FUNCTION_BLOCK MoveAbsoluteTask EXTENDS TcoCore.TcoTask IMPLEMENTS ITcoDriveSimple
VAR
    {attribute addProperty Name "<#Position#>"}
    _position : LREAL;
    {attribute addProperty Name "<#Velocity#>"}
    _velocity : LREAL;
    {attribute addProperty Name "<#Acceleration#>"}
    _acceleration : LREAL;
    {attribute addProperty Name "<#Deceleration#>"}
    _deceleration : LREAL;
    {attribute addProperty Name "<#Jerk#>"}
    _jerk : LREAL;
END_VAR
VAR
    {attribute 'hide'}
    _axisRef : REFERENCE TO TcoAxisRef;
    {attribute 'hide'}
    _mcMoveAbsolute : Tc2_MC2.MC_MoveAbsolute;
    {attribute 'hide'}
    _mcMoveAbsolutePreconditionOK : BOOL;
    {attribute 'hide'}
	_mcReadAxisEncoderReferenceSystem : MC_ReadParameter;
	
	_AxisEncoderReferenceSystem : eAxisEncoderReferenceSystem;
END_VAR

IF NOT __ISVALIDREF(_axisRef) THEN
    IF __ISVALIDREF(DriveRef) THEN
        _axisRef REF= DriveRef.AxisRef;
    ELSE
        RETURN;
    END_IF
END_IF

IF Execute() THEN
    _mcReadAxisEncoderReferenceSystem(Axis := _axisRef,
        Enable := TRUE,
        ParameterNumber := eAxisParameter.AxisEncoderReferenceSystem,
        ReadMode := Tc2_MC2.E_ReadMode.READMODE_ONCE);

    IF _mcReadAxisEncoderReferenceSystem.Valid THEN
        LREAL_TO_Tco_AxisEncoderReferenceSystem(_mcReadAxisEncoderReferenceSystem.Value, _AxisEncoderReferenceSystem);

        IF _AxisEncoderReferenceSystem = eAxisEncoderReferenceSystem.ABSOLUTE OR
            _AxisEncoderReferenceSystem = eAxisEncoderReferenceSystem.ABSOLUTE_MODULO OR
            _AxisEncoderReferenceSystem = eAxisEncoderReferenceSystem.ABSOLUTE_MULTITURN OR
            _AxisEncoderReferenceSystem = eAxisEncoderReferenceSystem.ABSOLUTE_SINGLETURN THEN
            _mcMoveAbsolutePreconditionOK := TRUE;
        ELSE
            _mcMoveAbsolutePreconditionOK := _axisRef.Status.Homed;
        END_IF
    END_IF

    IF NOT DriveRef._movementState.MovePreconditionsOk(THIS^, _mcMoveAbsolutePreconditionOK) THEN
        IF _mcReadAxisEncoderReferenceSystem.Valid AND NOT _mcMoveAbsolutePreconditionOK THEN
            Messenger.Error('Move absolute not possible as axis is Incremental and not Homed');
        END_IF

        RETURN;
    END_IF

    _mcMoveAbsolute(Axis := _axisRef,
        Execute := NOT _mcMoveAbsolute.Busy,
        Position := _position,
        Velocity := _velocity,
        Acceleration := _acceleration,
        Deceleration := _deceleration,
        Jerk := _jerk,
        BufferMode := Tc2_MC2.MC_Aborting,
        Done =>,
        Busy =>,
        Active =>,
        CommandAborted =>,
        Error =>,
        ErrorID =>);

    IF _mcMoveAbsolute.CommandAborted THEN
        THIS^.Abort();
    END_IF

    DoneWhen(_mcMoveAbsolute.Done);
    ThrowWhen(_mcMoveAbsolute.Error);
END_IF

PROPERTY DriveRef : REFERENCE TO TcoDriveSimple
GET
VAR
    _drive : ITcoDriveSimple := 0;
END_VAR
IF __QUERYINTERFACE(THIS^.Parent, _drive) THEN
    DriveRef REF= _drive.DriveRef;
END_IF
END_GET
END_PROPERTY

METHOD PUBLIC FB_init : BOOL
VAR_INPUT
    bInitRetains : BOOL; // if TRUE, the retain variables are initialized (warm start / cold start)
    bInCopyCode : BOOL; // if TRUE, the instance afterwards gets moved into the copy code (online change)
  	ParentObject : ITcoObject;	
END_VAR
END_METHOD

METHOD INTERNAL InvokeWithParams : ITcoTaskStatus
VAR_INPUT
    inPosition : LREAL;
    inVelocity : LREAL;
    inAcceleration : LREAL;
    inDeceleration : LREAL;
    inJerk : LREAL;
END_VAR
_position := inPosition;
_velocity := inVelocity;
_acceleration := inAcceleration;
_deceleration := inDeceleration;
_jerk := inJerk;
InvokeWithParams := THIS^.Invoke();
END_METHOD

(*~
	<docu>
		<summary>
			Executes when task is aborted.
		</summary>			
	</docu>	
~*)
METHOD PROTECTED OnAbort
IF NOT __ISVALIDREF(_axisRef) THEN
    IF __ISVALIDREF(DriveRef) THEN
        _axisRef REF= DriveRef.AxisRef;
    ELSE
        RETURN;
    END_IF
END_IF

THIS^.DriveRef.Stop(-1, -1);
_mcMoveAbsolute(Axis := _axisRef, Execute := FALSE);
_mcReadAxisEncoderReferenceSystem(Axis :=_axisRef,Enable := FALSE);
THIS^.DriveRef._movementState.Restore();
END_METHOD

(*~
	<docu>
		<summary>
			Executes when task reaches the ```Done``` state .
		</summary>			
	</docu>	
~*)
METHOD PROTECTED OnDone
_mcMoveAbsolute(Axis := _axisRef, Execute := FALSE);
_mcReadAxisEncoderReferenceSystem(Axis :=_axisRef,Enable := FALSE);
THIS^.DriveRef._movementState.Restore();
END_METHOD

(*~
	<docu>
		<summary>
			Executes when task reaches the ```Error``` state.
			<para>
				Do not confuse with <see cref="PlcDocu.TcoCore.TcoTask.WhileError()"/>, that is called cyclically until '''Error''' state is left.
			</para>
		</summary>			
	</docu>	
~*)
METHOD PROTECTED OnError
THIS^.DriveRef._movementState.Restore();

IF NOT _axisRef.Status.Error THEN
	DriveRef.SetErrorID( DriveRef._moveAbsoluteTask._mcMoveAbsolute.ErrorID);
END_IF
_mcMoveAbsolute(Axis := _axisRef, Execute := FALSE);
_mcReadAxisEncoderReferenceSystem(Axis :=_axisRef,Enable := FALSE);
END_METHOD

METHOD PROTECTED OnStart
_mcMoveAbsolute(Axis := _axisRef, Execute := FALSE);
_mcReadAxisEncoderReferenceSystem(Axis :=_axisRef,Enable := FALSE);
END_METHOD

(*~
	<docu>
		<summary>
			Restores this instance to the Ready state. Can be called explicitly or from within one of the restore mechanisms.
			<para>
				See also <see cref="PlcDocu.TcoCore.TcoTask.AutoRestorable()"/>
			</para>
		</summary>			
	</docu>	
~*)
METHOD Restore : ITcoRestorable
SUPER^.Restore();
END_METHOD

(*~
	<docu>
		<summary>
			Executes until task is in ```Error``` state .
		</summary>			
	</docu>	
~*)
METHOD PROTECTED WhileError
IF NOT _axisRef.Status.Error THEN
	DriveRef.SetErrorID( DriveRef._moveAbsoluteTask._mcMoveAbsolute.ErrorID);
    _mcMoveAbsolute(Axis := _axisRef, Execute := FALSE);
END_IF
END_METHOD

END_FUNCTION_BLOCK

(* stored: Version 1.1.0.1, ProductVersion 3.1.4024.12
   POU MoveAbsoluteTask: Id {8ec2cded-bd2e-0780-1c2c-713ba1fe9cfc}, SpecialFunc None
   Property DriveRef: Id {c918ab99-0887-0ba7-3e18-f42d76a60832}
   Get Get: Id {6cdc2aba-e2cc-09b5-2389-125dc9763c8c}
   Method FB_init: Id {0d82c97d-0789-05e0-17e6-78c74f6d4a10}
   Method InvokeWithParams: Id {831dee00-d9fb-0de4-16b7-4a6a3ef02f08}
   Method OnAbort: Id {31011d7c-432f-0571-1b49-be504ea7c23d}
   Method OnDone: Id {223dc89a-9f91-000c-1309-16f5f6432081}
   Method OnError: Id {ab9dc157-8d3b-0fc7-39e0-f7e22d57a5d0}
   Method OnStart: Id {1491f5ba-9f11-0ec9-2ca9-fc10d819bac1}
   Method Restore: Id {6b9c9854-0555-0eef-069a-af2d2447715a}
   Method WhileError: Id {efa8f938-4579-0e7b-3fc7-36ccb3207ab2} *)
